ABB RobotStudio station: Robogrammetry.rsstn

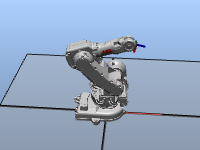
Station Robogrammetry (saved by RobotStudio 7.0.8504.151)
Controller IRB_140T_6kg_0.81m
  mechanical unit ROB_1: IRB140T_6_81_C_03, 6 joints, base frame (0, 0, 0) mm
Layout (positions relative to the parent item):
  - IRB140T_6_81_C_03 [mechanism, from Robots\IRB140T_6_81_C_G_03.rslib] at (0, 0, 0) mm; joint values [0.0696, -0.8196, 0.5372, 0, 0.5236, 0] (rad or m)
